PROGRAM main
VAR
    CountDown AT %QX0.0 : BOOL;
    LoadCounter AT %QX0.1 : BOOL;
    Done AT %QX0.2 : BOOL;
    CurrentCount AT %MD0 : DINT;
    CounterInstance : CTD_DINT;
    Preset : DINT := 3;
END_VAR

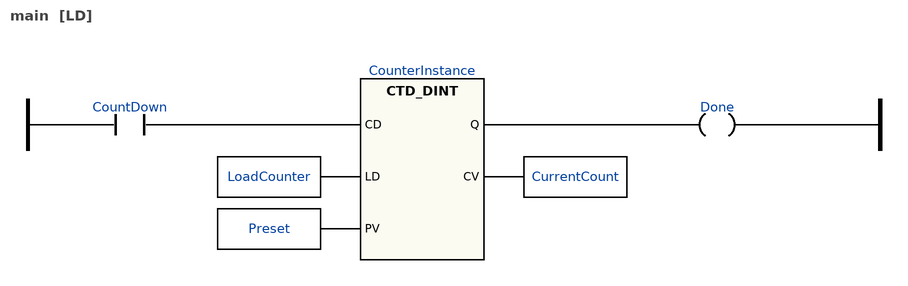
(* LD diagram, written out as Structured Text *)
CounterInstance(CD := CountDown, LD := LoadCounter, PV := Preset);
Done := CounterInstance.Q;
CurrentCount := CounterInstance.CV;
END_PROGRAM
